// SIMATIC S7-200 SMART project (STEP 7-Micro/WIN SMART), CPU SR40

SYMBOL_TABLE 系统符号
Always_On        SM0.0    // 始终接通
END_SYMBOL_TABLE

ORGANIZATION_BLOCK MAIN:OB1
TITLE=程序注释
BEGIN
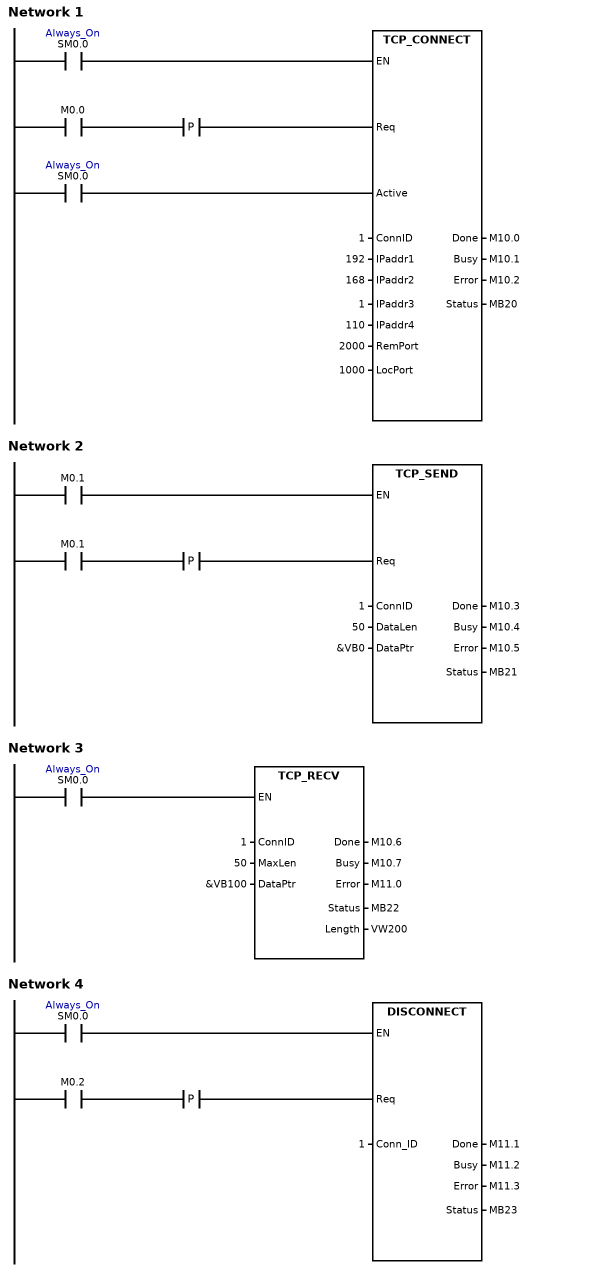
Network 1
LD     Always_On:SM0.0
=      L60.0
LD     M0.0
EU
=      L63.7
LD     Always_On:SM0.0
=      L63.6
LD     L60.0
CALL   TCP_CONNECT:SBR1, L63.7, L63.6, 1, 192, 168, 1, 110, 2000, 1000, M10.0, M10.1, M10.2, MB20
Network 2
LD     M0.1
=      L60.0
LD     M0.1
EU
=      L63.7
LD     L60.0
CALL   TCP_SEND:SBR2, L63.7, 1, 50, &VB0, M10.3, M10.4, M10.5, MB21
Network 3
LD     Always_On:SM0.0
CALL   TCP_RECV:SBR3, 1, 50, &VB100, M10.6, M10.7, M11.0, MB22, VW200
Network 4
LD     Always_On:SM0.0
=      L60.0
LD     M0.2
EU
=      L63.7
LD     L60.0
CALL   DISCONNECT:SBR4, L63.7, 1, M11.1, M11.2, M11.3, MB23
END_ORGANIZATION_BLOCK

// SBR1: protected block, not included

// SBR2: protected block, not included

// SBR3: protected block, not included

// SBR4: protected block, not included
